FUNCTION ModbusToReal : REAL
VAR_INPUT
	wHi : WORD;
    wLo : WORD;
END_VAR
VAR
	
	 dw : DWORD;
	 rR  : REAL;
END_VAR

// złożenie 2xWORD -> 32-bit (Big-Endian: HI potem LO)
dw := SHL(WORD_TO_DWORD(wHi), 16) OR WORD_TO_DWORD(wLo);

// reinterpretacja bitów DWORD jako REAL
MEMCPY(ADR(rR), ADR(dw), SIZEOF(rR));

ModbusToReal := rR;

END_FUNCTION

(* stored: Version 1.1.0.1, ProductVersion 3.1.4024.15
   POU ModbusToReal: Id {beda0692-9542-4cc6-98a2-158817cecd56}, SpecialFunc None *)
